PROGRAM MAIN
VAR
END_VAR

END_PROGRAM

(* stored: Version 1.1.0.1
   POU MAIN: Id {8c9d9970-7f52-426d-9820-70dfcef0beff} *)
